Staubli VAL3: status.pgx

program status()
  local num count
  local string callStack
  local string library
  local string program
  local num line
  local string code
begin
    //
  //\var count
  //\var callStack
  //\var library
  //\var program
  //\var line
  //\var code
  //
while true
    count=$taskCallStack(sTaskName[1],callStack)
    call parseStackInfo(callStack,library,program,line,code)
    if program=="SP_Traj"
      call list:resizeString(programList,max(size(programList),line))
      programList[line]=code
    endIf
  endWhile
end
